FUNCTION_BLOCK MainStation EXTENDS TcoCore.TcoObject
VAR
    turckRfidHead : RfidHead(THIS^, T#1MS);
    sUId          : T_MaxString;
END_VAR
VAR
        _uid          : BOOL;
END_VAR

turckRfidHead();

IF _uid THEN
    turckRfidHead.ReadUidMethod();
    _uid := FALSE;
END_IF

IF turckRfidHead.ReadUidTask.Done then
    sUId := turckRfidHead.sUId;
END_IF

END_FUNCTION_BLOCK

(* stored: Version 1.1.0.1, ProductVersion 3.1.4024.12
   POU MainStation: Id {aba662ba-0104-0d8c-3ede-cc6ee7a38896}, SpecialFunc None *)
